FUNCTION POU : BOOL
VAR_INPUT
 Tijd : TIME;
 Afstand : INT;
END_VAR
VAR
	TijdInSeconden : REAL;
	TransportbandSnelheid : REAL;
END_VAR

TijdInSeconden := TIME_TO_REAL(Tijd)/1000; // Zet de tijd om naar een REAL waarde in seconden

IF Afstand = 0 THEN // Controleer of de afstand gelijk is aan 0
    GVL.TransportBandSnelheid := 0; // Stel de transportbandsnelheid in op 0
ELSE	
    GVL.TransportBandSnelheid := Afstand / TijdInSeconden; // Bereken de snelheid van het transportband
END_IF

END_FUNCTION

(* stored: Version 1.1.0.1, ProductVersion 3.1.4024.12
   POU POU: Id {9a9488f8-69a9-4e57-85fd-b9790f2a86a4}, SpecialFunc None *)
